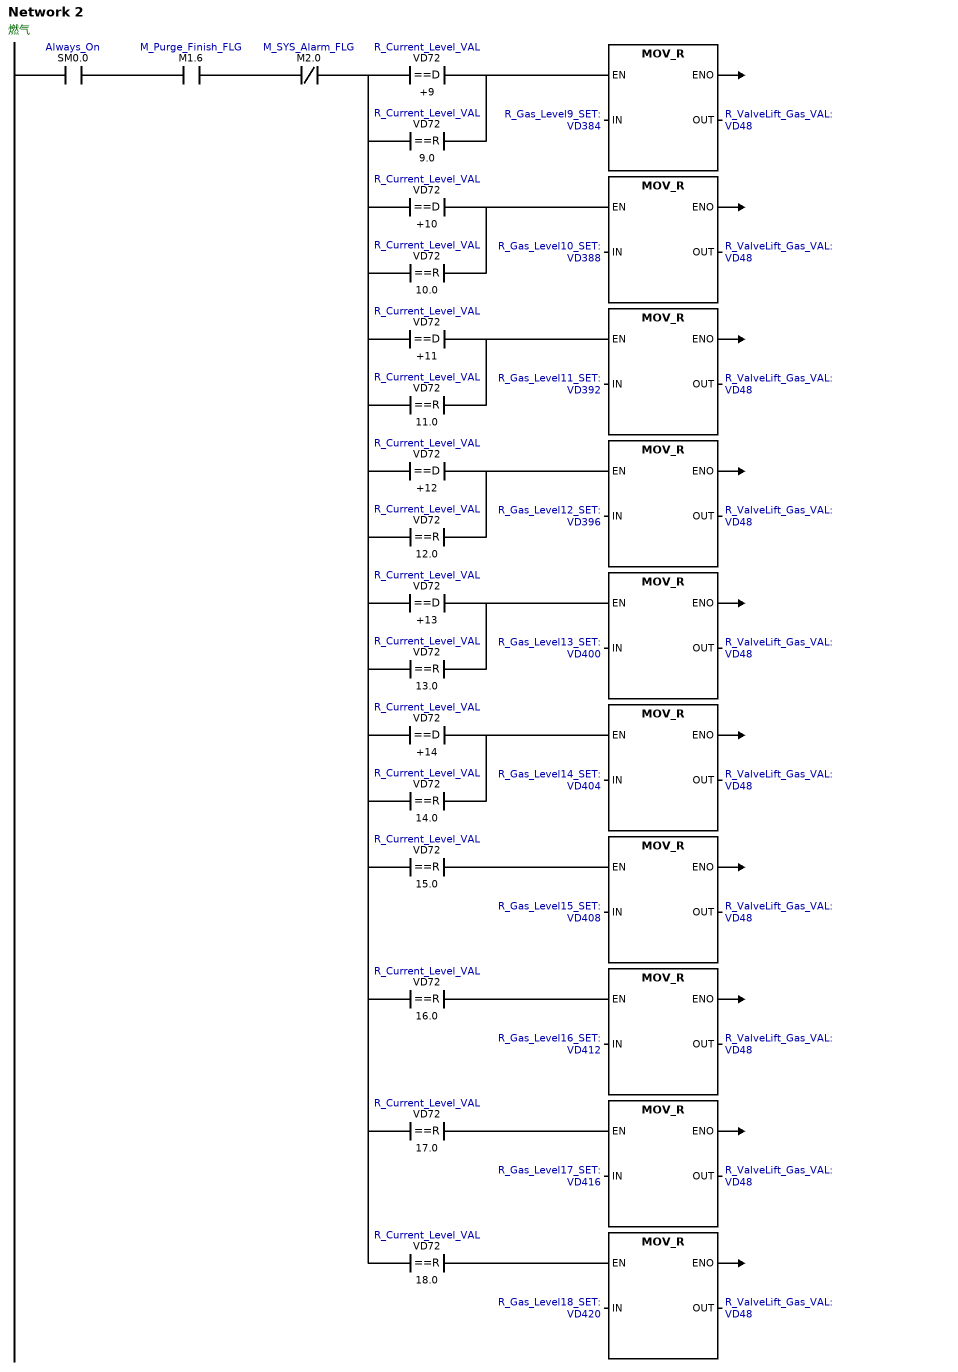
[picture p24: SBR6 networks 2-2]
Network 2
// 燃气
LD     Always_On:SM0.0
A      M_Purge_Finish_FLG:M1.6
AN     M_SYS_Alarm_FLG:M2.0
LPS
LDD=   R_Current_Level_VAL:VD72, +9
OR=    R_Current_Level_VAL:VD72, 9.0
ALD
MOVR   R_Gas_Level9_SET:VD384, R_ValveLift_Gas_VAL:VD48
LRD
LDD=   R_Current_Level_VAL:VD72, +10
OR=    R_Current_Level_VAL:VD72, 10.0
ALD
MOVR   R_Gas_Level10_SET:VD388, R_ValveLift_Gas_VAL:VD48
LRD
LDD=   R_Current_Level_VAL:VD72, +11
OR=    R_Current_Level_VAL:VD72, 11.0
ALD
MOVR   R_Gas_Level11_SET:VD392, R_ValveLift_Gas_VAL:VD48
LRD
LDD=   R_Current_Level_VAL:VD72, +12
OR=    R_Current_Level_VAL:VD72, 12.0
ALD
MOVR   R_Gas_Level12_SET:VD396, R_ValveLift_Gas_VAL:VD48
LRD
LDD=   R_Current_Level_VAL:VD72, +13
OR=    R_Current_Level_VAL:VD72, 13.0
ALD
MOVR   R_Gas_Level13_SET:VD400, R_ValveLift_Gas_VAL:VD48
LRD
LDD=   R_Current_Level_VAL:VD72, +14
OR=    R_Current_Level_VAL:VD72, 14.0
ALD
MOVR   R_Gas_Level14_SET:VD404, R_ValveLift_Gas_VAL:VD48
LPP
LPS
AR=    R_Current_Level_VAL:VD72, 15.0
MOVR   R_Gas_Level15_SET:VD408, R_ValveLift_Gas_VAL:VD48
LRD
AR=    R_Current_Level_VAL:VD72, 16.0
MOVR   R_Gas_Level16_SET:VD412, R_ValveLift_Gas_VAL:VD48
LRD
AR=    R_Current_Level_VAL:VD72, 17.0
MOVR   R_Gas_Level17_SET:VD416, R_ValveLift_Gas_VAL:VD48
LPP
AR=    R_Current_Level_VAL:VD72, 18.0
MOVR   R_Gas_Level18_SET:VD420, R_ValveLift_Gas_VAL:VD48
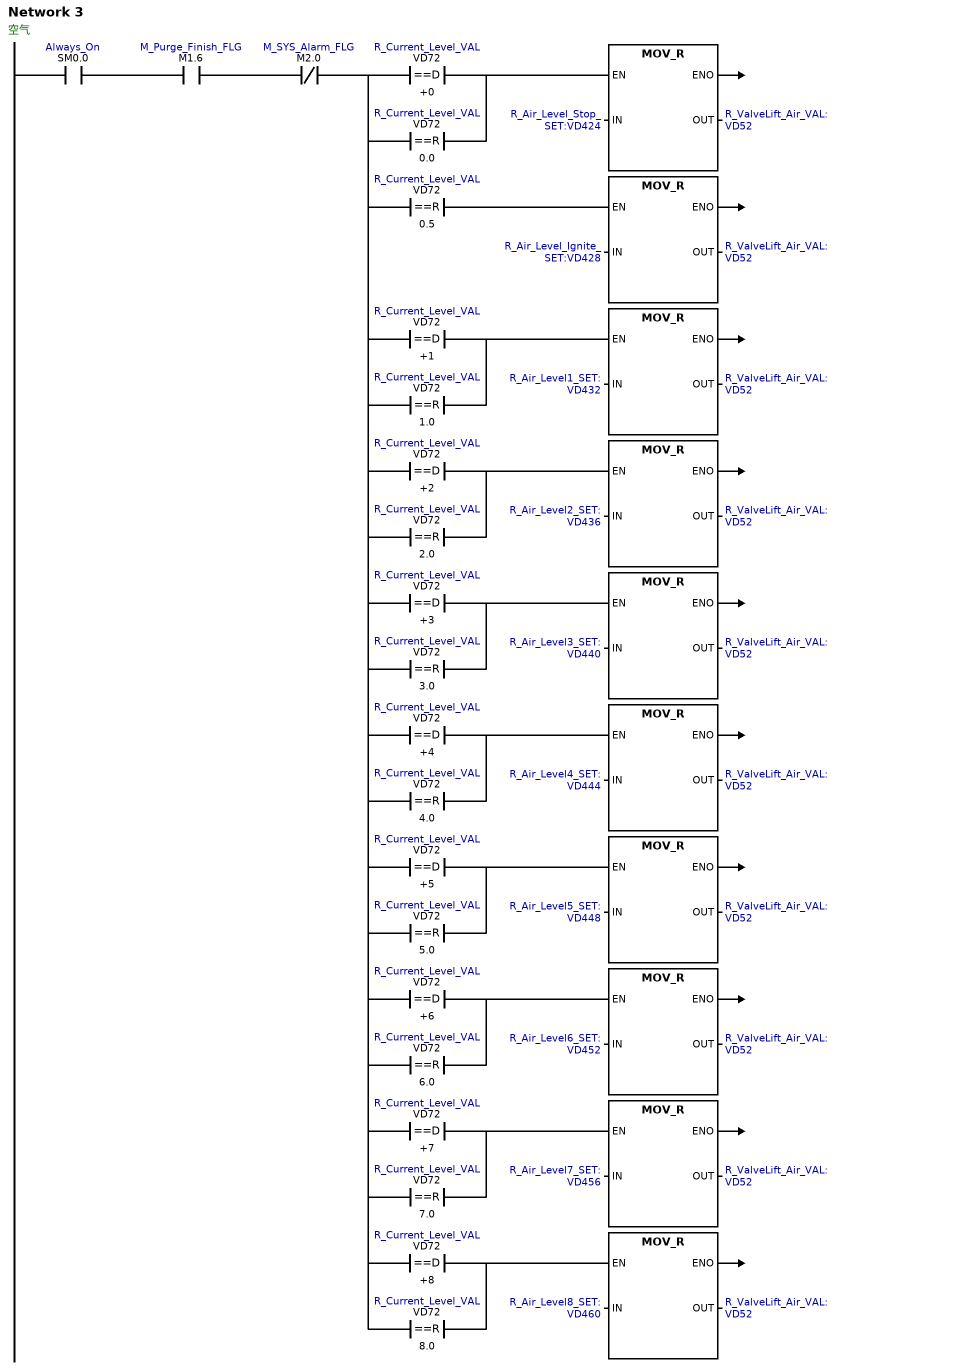
Network 3
// 空气
LD     Always_On:SM0.0
A      M_Purge_Finish_FLG:M1.6
AN     M_SYS_Alarm_FLG:M2.0
LPS
LDD=   R_Current_Level_VAL:VD72, +0
OR=    R_Current_Level_VAL:VD72, 0.0
ALD
MOVR   R_Air_Level_Stop_SET:VD424, R_ValveLift_Air_VAL:VD52
LRD
AR=    R_Current_Level_VAL:VD72, 0.5
MOVR   R_Air_Level_Ignite_SET:VD428, R_ValveLift_Air_VAL:VD52
LRD
LDD=   R_Current_Level_VAL:VD72, +1
OR=    R_Current_Level_VAL:VD72, 1.0
ALD
MOVR   R_Air_Level1_SET:VD432, R_ValveLift_Air_VAL:VD52
LRD
LDD=   R_Current_Level_VAL:VD72, +2
OR=    R_Current_Level_VAL:VD72, 2.0
ALD
MOVR   R_Air_Level2_SET:VD436, R_ValveLift_Air_VAL:VD52
LRD
LDD=   R_Current_Level_VAL:VD72, +3
OR=    R_Current_Level_VAL:VD72, 3.0
ALD
MOVR   R_Air_Level3_SET:VD440, R_ValveLift_Air_VAL:VD52
LRD
LDD=   R_Current_Level_VAL:VD72, +4
OR=    R_Current_Level_VAL:VD72, 4.0
ALD
MOVR   R_Air_Level4_SET:VD444, R_ValveLift_Air_VAL:VD52
LRD
LDD=   R_Current_Level_VAL:VD72, +5
OR=    R_Current_Level_VAL:VD72, 5.0
ALD
MOVR   R_Air_Level5_SET:VD448, R_ValveLift_Air_VAL:VD52
LRD
LDD=   R_Current_Level_VAL:VD72, +6
OR=    R_Current_Level_VAL:VD72, 6.0
ALD
MOVR   R_Air_Level6_SET:VD452, R_ValveLift_Air_VAL:VD52
LRD
LDD=   R_Current_Level_VAL:VD72, +7
OR=    R_Current_Level_VAL:VD72, 7.0
ALD
MOVR   R_Air_Level7_SET:VD456, R_ValveLift_Air_VAL:VD52
LPP
LDD=   R_Current_Level_VAL:VD72, +8
OR=    R_Current_Level_VAL:VD72, 8.0
ALD
MOVR   R_Air_Level8_SET:VD460, R_ValveLift_Air_VAL:VD52
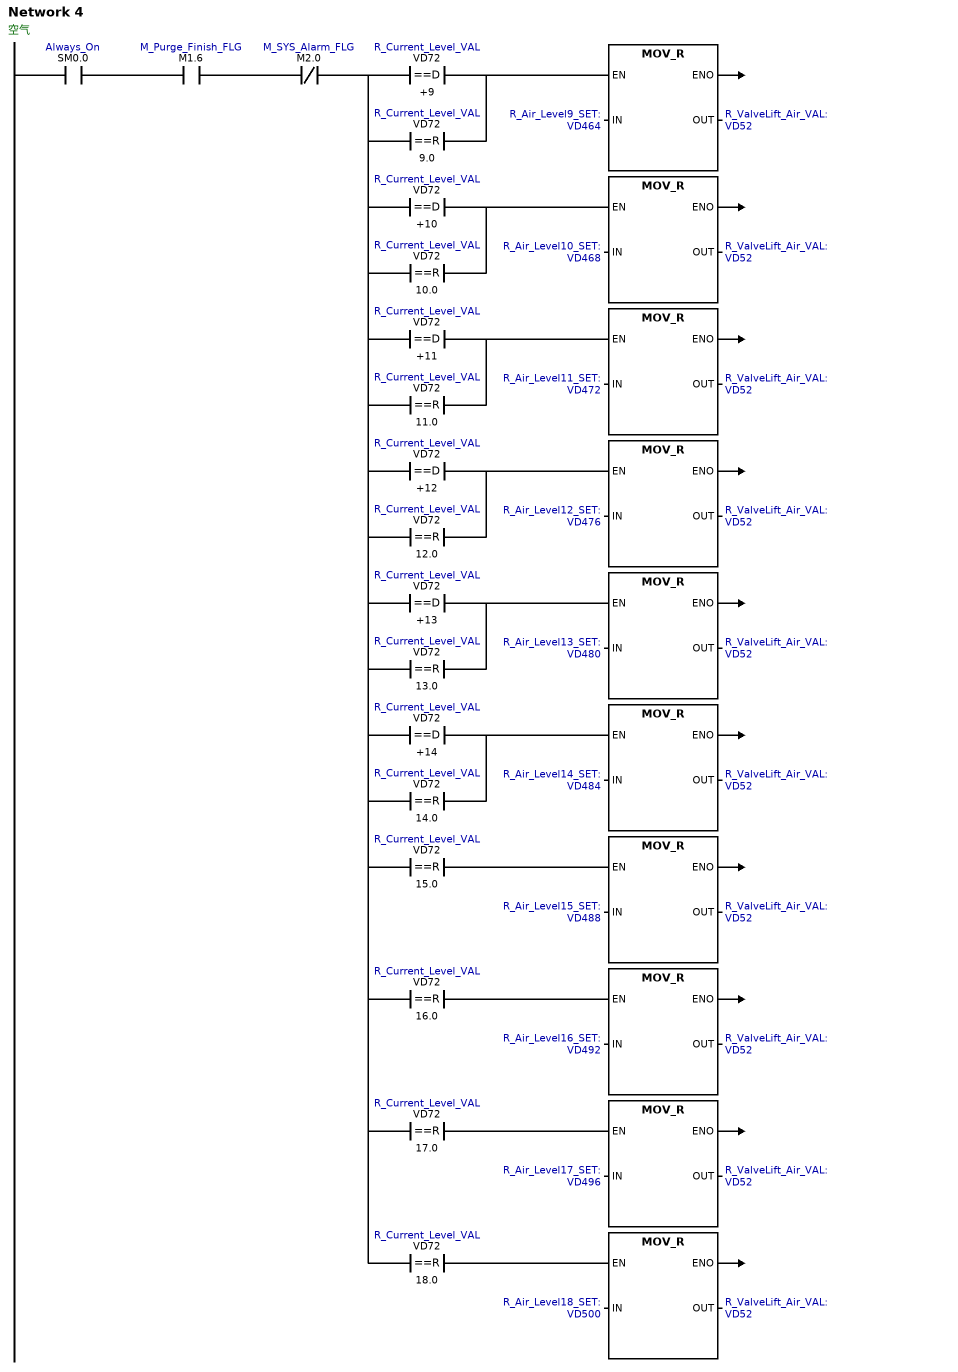
Network 4
// 空气
LD     Always_On:SM0.0
A      M_Purge_Finish_FLG:M1.6
AN     M_SYS_Alarm_FLG:M2.0
LPS
LDD=   R_Current_Level_VAL:VD72, +9
OR=    R_Current_Level_VAL:VD72, 9.0
ALD
MOVR   R_Air_Level9_SET:VD464, R_ValveLift_Air_VAL:VD52
LRD
LDD=   R_Current_Level_VAL:VD72, +10
OR=    R_Current_Level_VAL:VD72, 10.0
ALD
MOVR   R_Air_Level10_SET:VD468, R_ValveLift_Air_VAL:VD52
LRD
LDD=   R_Current_Level_VAL:VD72, +11
OR=    R_Current_Level_VAL:VD72, 11.0
ALD
MOVR   R_Air_Level11_SET:VD472, R_ValveLift_Air_VAL:VD52
LRD
LDD=   R_Current_Level_VAL:VD72, +12
OR=    R_Current_Level_VAL:VD72, 12.0
ALD
MOVR   R_Air_Level12_SET:VD476, R_ValveLift_Air_VAL:VD52
LRD
LDD=   R_Current_Level_VAL:VD72, +13
OR=    R_Current_Level_VAL:VD72, 13.0
ALD
MOVR   R_Air_Level13_SET:VD480, R_ValveLift_Air_VAL:VD52
LRD
LDD=   R_Current_Level_VAL:VD72, +14
OR=    R_Current_Level_VAL:VD72, 14.0
ALD
MOVR   R_Air_Level14_SET:VD484, R_ValveLift_Air_VAL:VD52
LPP
LPS
AR=    R_Current_Level_VAL:VD72, 15.0
MOVR   R_Air_Level15_SET:VD488, R_ValveLift_Air_VAL:VD52
LRD
AR=    R_Current_Level_VAL:VD72, 16.0
MOVR   R_Air_Level16_SET:VD492, R_ValveLift_Air_VAL:VD52
LRD
AR=    R_Current_Level_VAL:VD72, 17.0
MOVR   R_Air_Level17_SET:VD496, R_ValveLift_Air_VAL:VD52
LPP
AR=    R_Current_Level_VAL:VD72, 18.0
MOVR   R_Air_Level18_SET:VD500, R_ValveLift_Air_VAL:VD52
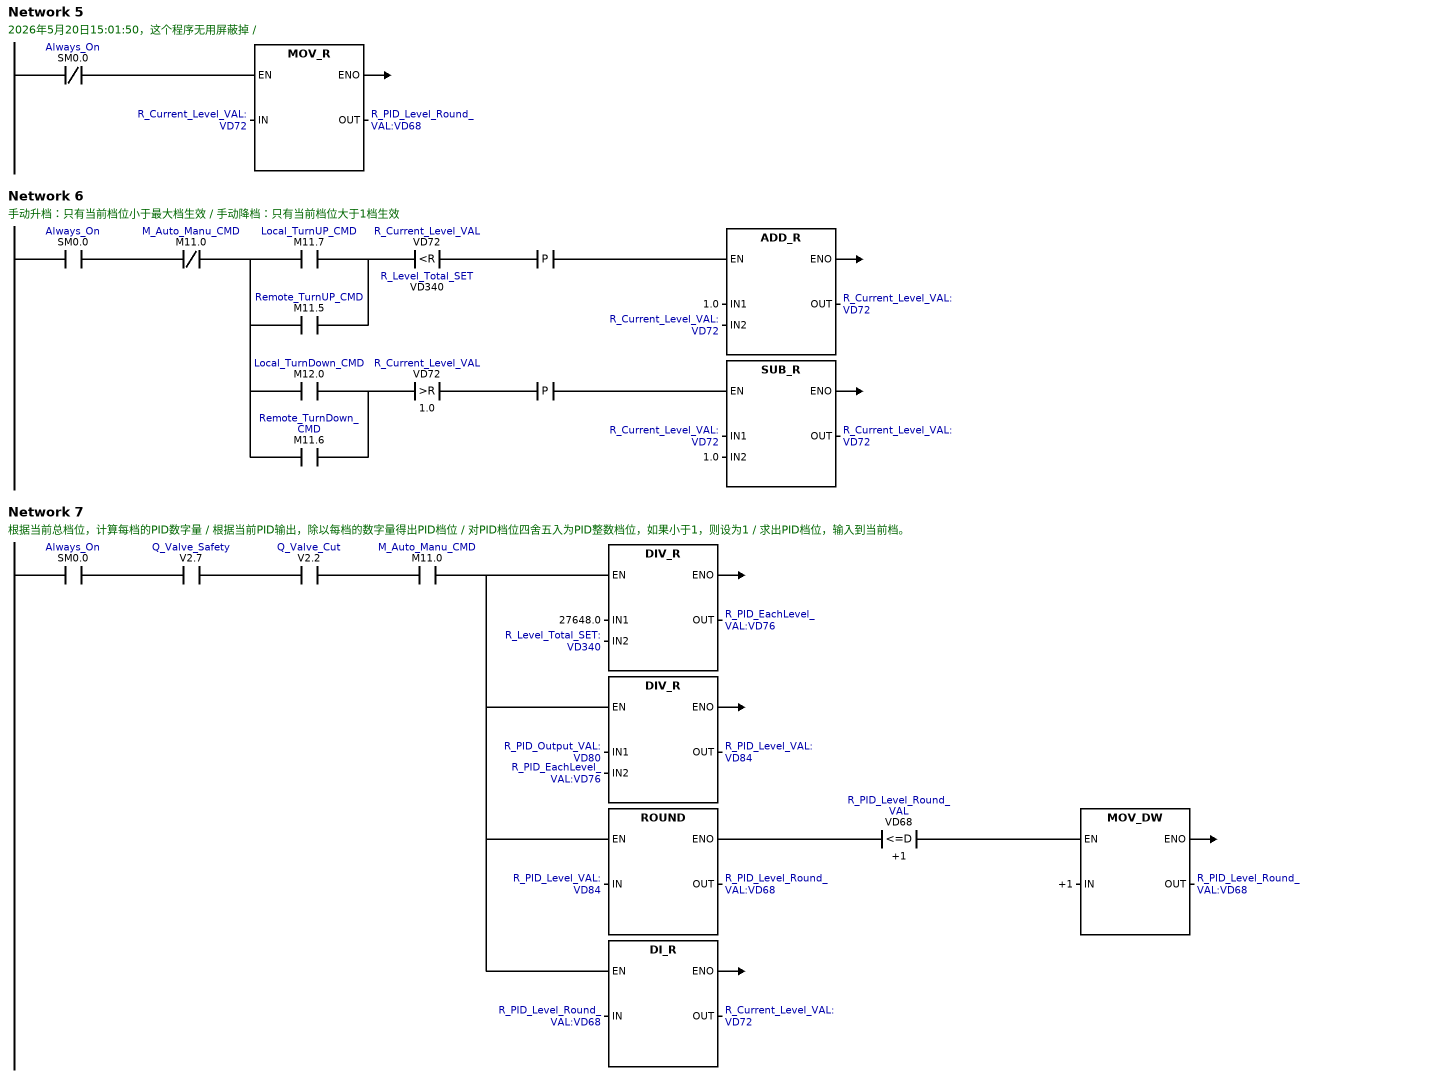
Network 5
// 2026年5月20日15:01:50，这个程序无用屏蔽掉
// 
LDN    Always_On:SM0.0
MOVR   R_Current_Level_VAL:VD72, R_PID_Level_Round_VAL:VD68
Network 6
// 手动升档：只有当前档位小于最大档生效
// 手动降档：只有当前档位大于1档生效
LD     Always_On:SM0.0
AN     M_Auto_Manu_CMD:M11.0
LPS
LD     Local_TurnUP_CMD:M11.7
O      Remote_TurnUP_CMD:M11.5
ALD
AR<    R_Current_Level_VAL:VD72, R_Level_Total_SET:VD340
EU
+R     1.0, R_Current_Level_VAL:VD72
LPP
LD     Local_TurnDown_CMD:M12.0
O      Remote_TurnDown_CMD:M11.6
ALD
AR>    R_Current_Level_VAL:VD72, 1.0
EU
-R     1.0, R_Current_Level_VAL:VD72
Network 7
// 根据当前总档位，计算每档的PID数字量
// 根据当前PID输出，除以每档的数字量得出PID档位
// 对PID档位四舍五入为PID整数档位，如果小于1，则设为1
// 求出PID档位，输入到当前档。
LD     Always_On:SM0.0
A      Q_Valve_Safety:V2.7
A      Q_Valve_Cut:V2.2
A      M_Auto_Manu_CMD:M11.0
LPS
MOVR   27648.0, R_PID_EachLevel_VAL:VD76
/R     R_Level_Total_SET:VD340, R_PID_EachLevel_VAL:VD76
MOVR   R_PID_Output_VAL:VD80, R_PID_Level_VAL:VD84
/R     R_PID_EachLevel_VAL:VD76, R_PID_Level_VAL:VD84
ROUND  R_PID_Level_VAL:VD84, R_PID_Level_Round_VAL:VD68
AENO
AD<=   R_PID_Level_Round_VAL:VD68, +1
MOVD   +1, R_PID_Level_Round_VAL:VD68
LPP
DTR    R_PID_Level_Round_VAL:VD68, R_Current_Level_VAL:VD72
END_SUBROUTINE_BLOCK

SUBROUTINE_BLOCK 远程通讯:SBR7
TITLE=远程通讯子程序
// 功能：
// 1、初始化从站（PLC）
// 	模式Mode（通讯协议）：	1、Modubs协议；0、PPI协
// 	地址Addr	：	1-247
// 	波特率Baud：	1200、2400、4800、9600、19200、38400、57600、11500
// 	奇偶校验Parity：	0无校验、1奇校验、2偶校验
// 	端口Port：	0=CPU集成RS-485端口，1=可选信号板上的RS-485或RS-232
// 	延时Delay：	可以是0-32767
// 	MaxIQ：		设置Modbus地址0XXXX和1XXXX可用 的I和Q点数，0-256
// 	MaxAI：		设置Modbus地址3XXXX可用的字输入（AI）寄存器数，0（CR系列）或56（其它系列）
// 	MaxHold：	设置Modbus地址4XXXX或4yyyyy可访问的V存储器中的字保持寄存器数。如果要允许 Modbus 主站访问 2000 个字节的 V 存储器，请将 MaxHold的值设置为 1000 个字（保持寄存器）
// 	HoldStart：	是 V 存储器中保持寄存器的起始地址	
// 
// 2、处理主站请求
// 在每次扫描处理主站请求
// 
// 
// 
// 3、显示设备状态：
// 	故障状态RTU
// 	自动状态RTU
// 	启动状态RTU
// 	停止状态RTU
// 	本地远程状态RTU
// 
// 4、处理DCS传送过来的温度数据,VW1898
BEGIN
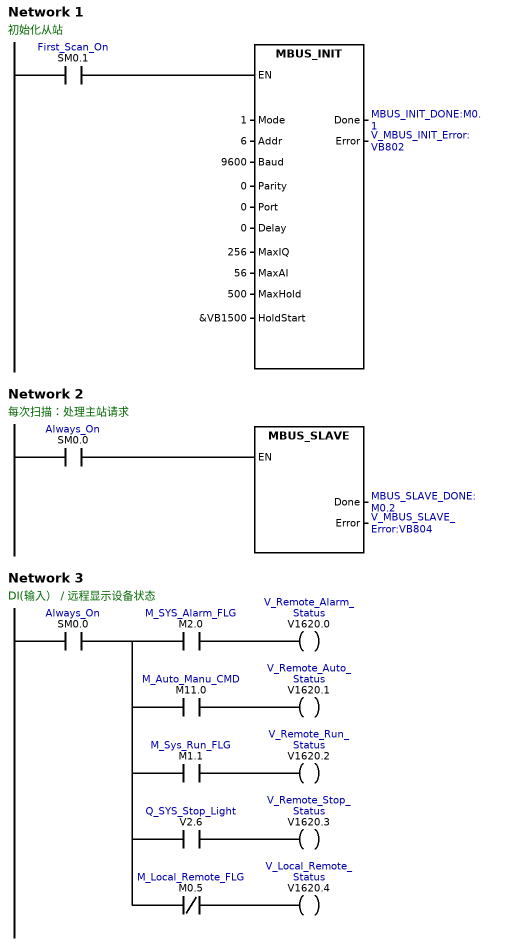
Network 1
// 初始化从站
LD     First_Scan_On:SM0.1
CALL   MBUS_INIT:SBR21, 1, 6, 9600, 0, 0, 0, 256, 56, 500, &VB1500, MBUS_INIT_DONE:M0.1, V_MBUS_INIT_Error:VB802
Network 2
// 每次扫描：处理主站请求
LD     Always_On:SM0.0
CALL   MBUS_SLAVE:SBR22, MBUS_SLAVE_DONE:M0.2, V_MBUS_SLAVE_Error:VB804
Network 3
// DI(输入）
// 远程显示设备状态
LD     Always_On:SM0.0
LPS
A      M_SYS_Alarm_FLG:M2.0
=      V_Remote_Alarm_Status:V1620.0
LRD
A      M_Auto_Manu_CMD:M11.0
=      V_Remote_Auto_Status:V1620.1
LRD
A      M_Sys_Run_FLG:M1.1
=      V_Remote_Run_Status:V1620.2
LRD
A      Q_SYS_Stop_Light:V2.6
=      V_Remote_Stop_Status:V1620.3
LPP
AN     M_Local_Remote_FLG:M0.5
=      V_Local_Remote_Status:V1620.4
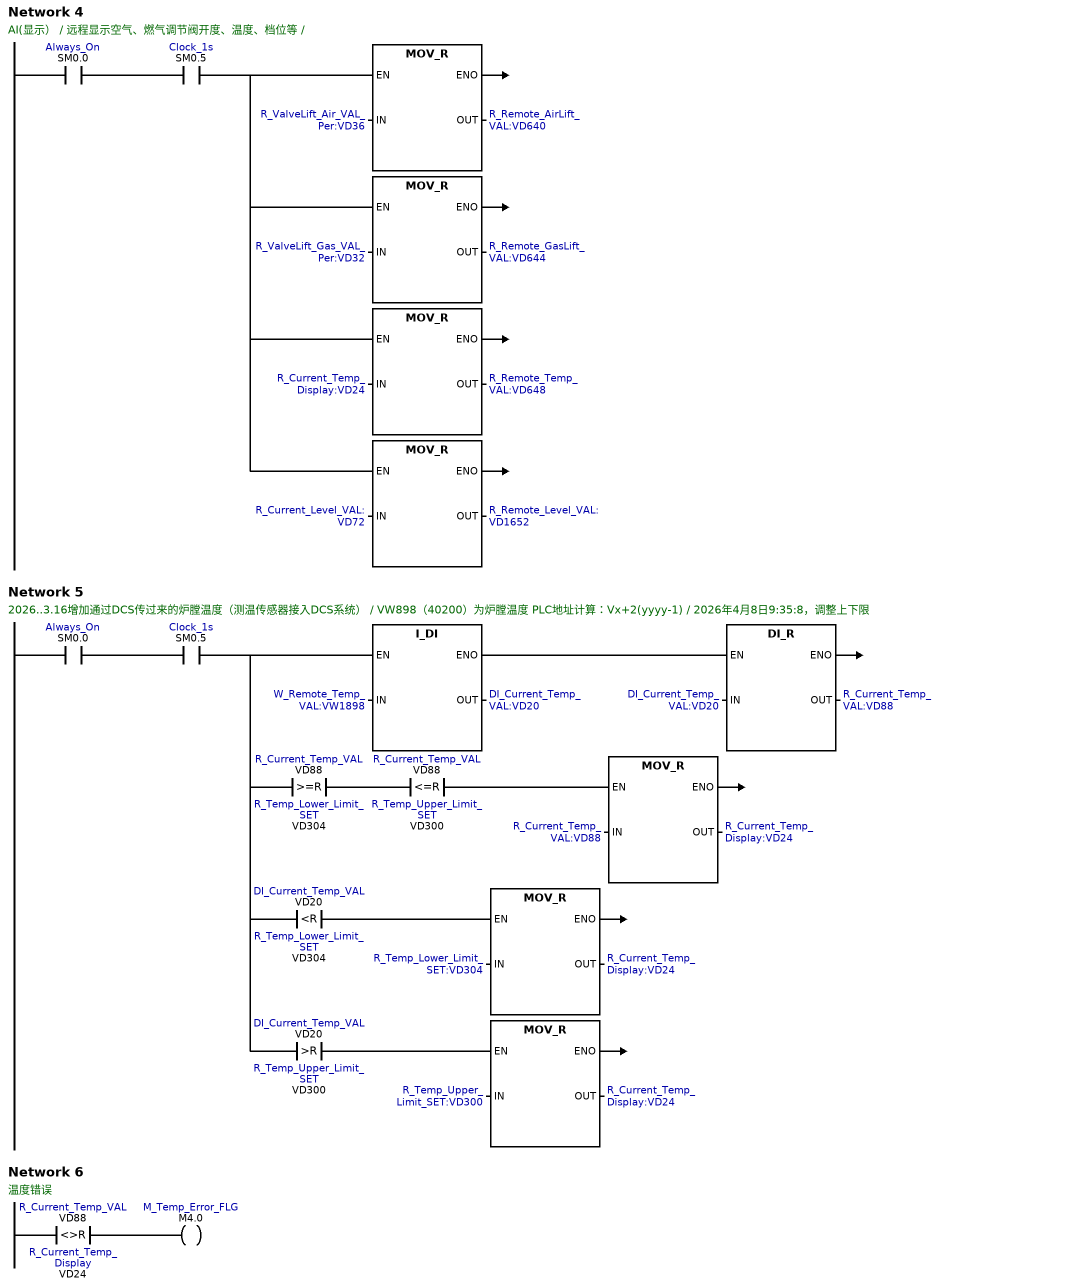
Network 4
// AI(显示）
// 远程显示空气、燃气调节阀开度、温度、档位等
// 
LD     Always_On:SM0.0
A      Clock_1s:SM0.5
MOVR   R_ValveLift_Air_VAL_Per:VD36, R_Remote_AirLift_VAL:VD640
MOVR   R_ValveLift_Gas_VAL_Per:VD32, R_Remote_GasLift_VAL:VD644
MOVR   R_Current_Temp_Display:VD24, R_Remote_Temp_VAL:VD648
MOVR   R_Current_Level_VAL:VD72, R_Remote_Level_VAL:VD1652
Network 5
// 2026..3.16增加通过DCS传过来的炉膛温度（测温传感器接入DCS系统）
// VW898（40200）为炉膛温度 PLC地址计算：Vx+2(yyyy-1)
// 2026年4月8日9:35:8，调整上下限
LD     Always_On:SM0.0
A      Clock_1s:SM0.5
LPS
ITD    W_Remote_Temp_VAL:VW1898, DI_Current_Temp_VAL:VD20
AENO
DTR    DI_Current_Temp_VAL:VD20, R_Current_Temp_VAL:VD88
LRD
AR>=   R_Current_Temp_VAL:VD88, R_Temp_Lower_Limit_SET:VD304
AR<=   R_Current_Temp_VAL:VD88, R_Temp_Upper_Limit_SET:VD300
MOVR   R_Current_Temp_VAL:VD88, R_Current_Temp_Display:VD24
LRD
AR<    DI_Current_Temp_VAL:VD20, R_Temp_Lower_Limit_SET:VD304
MOVR   R_Temp_Lower_Limit_SET:VD304, R_Current_Temp_Display:VD24
LPP
AR>    DI_Current_Temp_VAL:VD20, R_Temp_Upper_Limit_SET:VD300
MOVR   R_Temp_Upper_Limit_SET:VD300, R_Current_Temp_Display:VD24
Network 6
// 温度错误
LDR<>  R_Current_Temp_VAL:VD88, R_Current_Temp_Display:VD24
=      M_Temp_Error_FLG:M4.0
END_SUBROUTINE_BLOCK

SUBROUTINE_BLOCK IO设备:SBR8
TITLE=子程序注释
// 1、IO映射
// 2、统一输出
// 	蜂鸣器
// 	点火阀
// 	主火阀V2
// 	点火变压器
// 	有火指示灯
// 	启动指示灯
// 	停止指示灯
// 	安全阀V1
// 
// 
BEGIN
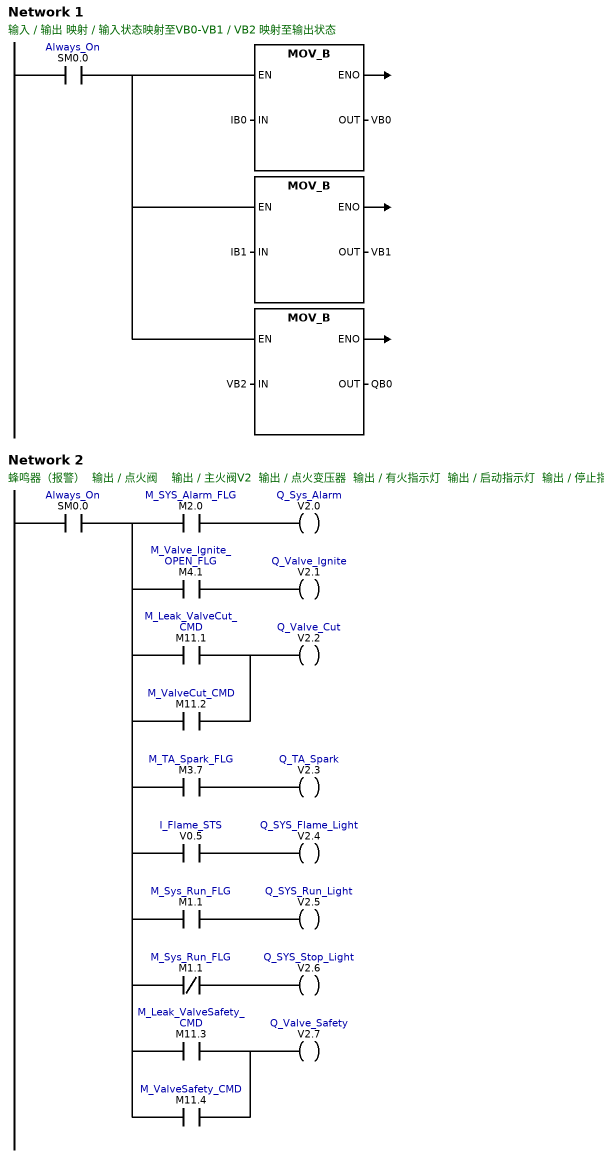
Network 1
// 输入 / 输出 映射
// 输入状态映射至VB0-VB1
// VB2 映射至输出状态
LD     Always_On:SM0.0
MOVB   IB0, VB0
MOVB   IB1, VB1
MOVB   VB2, QB0
Network 2
// 蜂鸣器（报警）	输出
// 点火阀		输出
// 主火阀V2	输出
// 点火变压器	输出
// 有火指示灯	输出
// 启动指示灯	输出
// 停止指示灯	输出
// 安全阀V1	输出
// 
LD     Always_On:SM0.0
LPS
A      M_SYS_Alarm_FLG:M2.0
=      Q_Sys_Alarm:V2.0
LRD
A      M_Valve_Ignite_OPEN_FLG:M4.1
=      Q_Valve_Ignite:V2.1
LRD
LD     M_Leak_ValveCut_CMD:M11.1
O      M_ValveCut_CMD:M11.2
ALD
=      Q_Valve_Cut:V2.2
LRD
LPS
A      M_TA_Spark_FLG:M3.7
=      Q_TA_Spark:V2.3
LRD
A      I_Flame_STS:V0.5
=      Q_SYS_Flame_Light:V2.4
LRD
A      M_Sys_Run_FLG:M1.1
=      Q_SYS_Run_Light:V2.5
LPP
AN     M_Sys_Run_FLG:M1.1
=      Q_SYS_Stop_Light:V2.6
LPP
LD     M_Leak_ValveSafety_CMD:M11.3
O      M_ValveSafety_CMD:M11.4
ALD
=      Q_Valve_Safety:V2.7
END_SUBROUTINE_BLOCK

SUBROUTINE_BLOCK 运行时间:SBR9
TITLE=
BEGIN
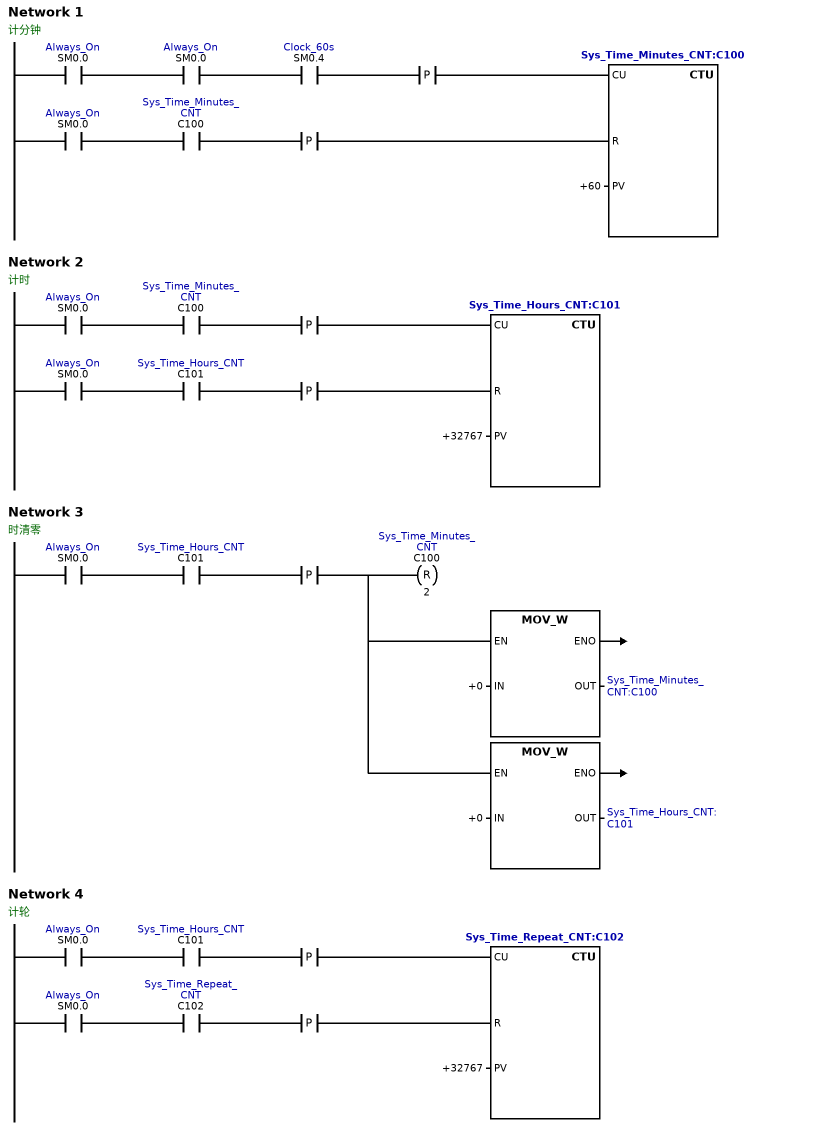
Network 1
// 计分钟
LD     Always_On:SM0.0
A      Always_On:SM0.0
A      Clock_60s:SM0.4
EU
LD     Always_On:SM0.0
A      Sys_Time_Minutes_CNT:C100
EU
CTU    Sys_Time_Minutes_CNT:C100, +60
Network 2
// 计时
LD     Always_On:SM0.0
A      Sys_Time_Minutes_CNT:C100
EU
LD     Always_On:SM0.0
A      Sys_Time_Hours_CNT:C101
EU
CTU    Sys_Time_Hours_CNT:C101, +32767
Network 3
// 时清零
LD     Always_On:SM0.0
A      Sys_Time_Hours_CNT:C101
EU
R      Sys_Time_Minutes_CNT:C100, 2
MOVW   +0, Sys_Time_Minutes_CNT:C100
MOVW   +0, Sys_Time_Hours_CNT:C101
Network 4
// 计轮
LD     Always_On:SM0.0
A      Sys_Time_Hours_CNT:C101
EU
LD     Always_On:SM0.0
A      Sys_Time_Repeat_CNT:C102
EU
CTU    Sys_Time_Repeat_CNT:C102, +32767
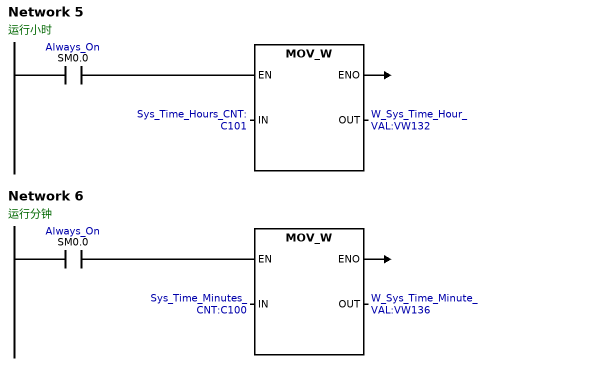
Network 5
// 运行小时
LD     Always_On:SM0.0
MOVW   Sys_Time_Hours_CNT:C101, W_Sys_Time_Hour_VAL:VW132
Network 6
// 运行分钟
LD     Always_On:SM0.0
MOVW   Sys_Time_Minutes_CNT:C100, W_Sys_Time_Minute_VAL:VW136
END_SUBROUTINE_BLOCK

SUBROUTINE_BLOCK 报警复位:SBR13
TITLE=报警复位子程序
// 功能：
// 1、报警逻辑
// 系统故障报警停机如：	
// 	检漏报警		停机
// 	空气压力低报警		停机
// 	燃气压力高报警		停机
// 	燃气压力低报警		停机
// 	点火前检测到火焰报警	停机
// 	点火失败报警		停机
// 	火焰丢失报警		停机
// 关闭所有燃气阀门：包括点火阀、主火阀、安全阀、
// 复位点火成功标志，
// 
// 调节阀故障只显示
// 	空气调节阀检测失败报警	提示
// 	燃气调节阀检测失败报警	提示
// 
// 
// 2、复位逻辑
// 复位7个故障，M20.1-M20.7
// 
// 两个调节阀故障，上电的时候才复位，这里不复位。
// 
// 
// 
BEGIN
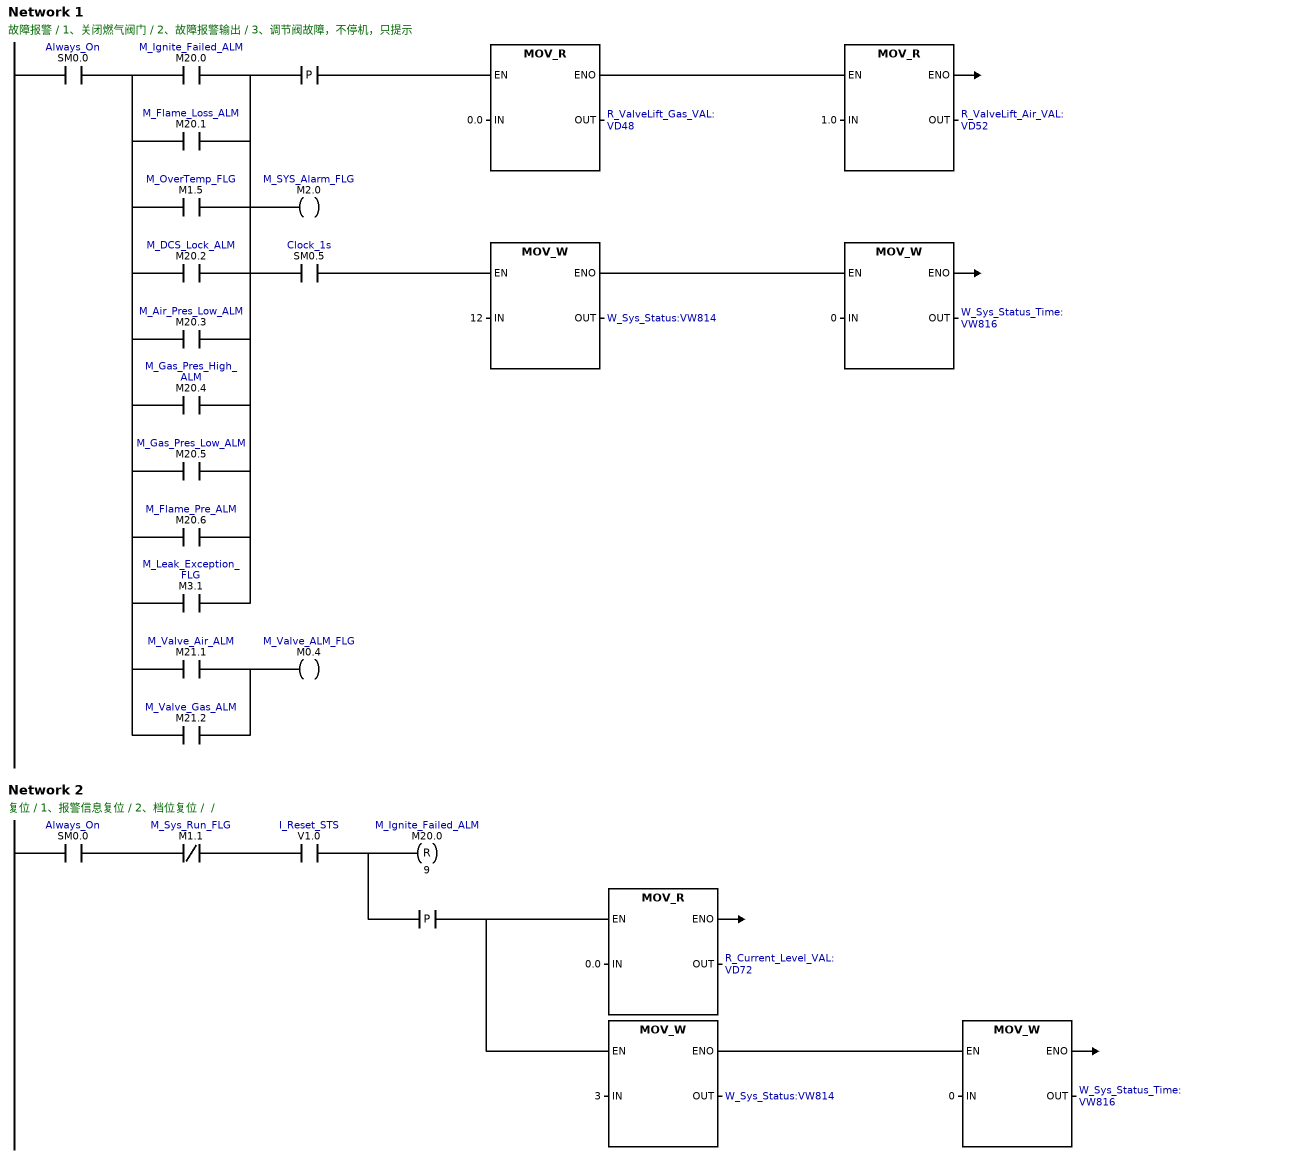
Network 1
// 故障报警
// 1、关闭燃气阀门
// 2、故障报警输出
// 3、调节阀故障，不停机，只提示
LD     Always_On:SM0.0
LPS
LD     M_Ignite_Failed_ALM:M20.0
O      M_Flame_Loss_ALM:M20.1
O      M_OverTemp_FLG:M1.5
O      M_DCS_Lock_ALM:M20.2
O      M_Air_Pres_Low_ALM:M20.3
O      M_Gas_Pres_High_ALM:M20.4
O      M_Gas_Pres_Low_ALM:M20.5
O      M_Flame_Pre_ALM:M20.6
O      M_Leak_Exception_FLG:M3.1
ALD
LPS
EU
MOVR   0.0, R_ValveLift_Gas_VAL:VD48
AENO
MOVR   1.0, R_ValveLift_Air_VAL:VD52
LRD
=      M_SYS_Alarm_FLG:M2.0
LPP
A      Clock_1s:SM0.5
MOVW   12, W_Sys_Status:VW814
AENO
MOVW   0, W_Sys_Status_Time:VW816
LPP
LD     M_Valve_Air_ALM:M21.1
O      M_Valve_Gas_ALM:M21.2
ALD
=      M_Valve_ALM_FLG:M0.4
Network 2
// 复位
// 1、报警信息复位
// 2、档位复位
// 
// 
LD     Always_On:SM0.0
AN     M_Sys_Run_FLG:M1.1
A      I_Reset_STS:V1.0
R      M_Ignite_Failed_ALM:M20.0, 9
EU
MOVR   0.0, R_Current_Level_VAL:VD72
MOVW   3, W_Sys_Status:VW814
AENO
MOVW   0, W_Sys_Status_Time:VW816
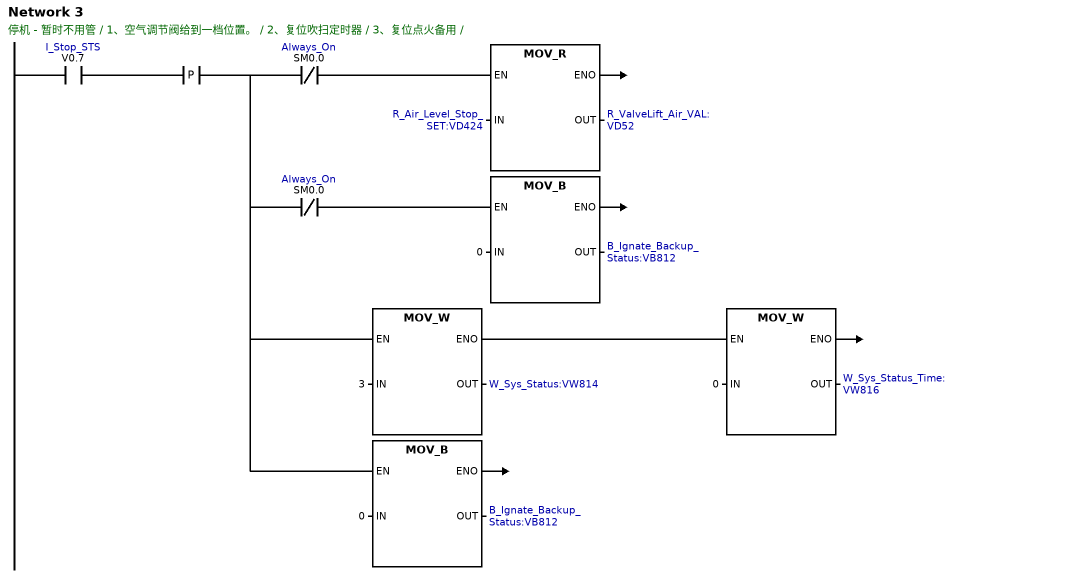
Network 3
// 停机 - 暂时不用管
// 1、空气调节阀给到一档位置。
// 2、复位吹扫定时器
// 3、复位点火备用
// 
LD     I_Stop_STS:V0.7
EU
LPS
AN     Always_On:SM0.0
MOVR   R_Air_Level_Stop_SET:VD424, R_ValveLift_Air_VAL:VD52
LRD
AN     Always_On:SM0.0
MOVB   0, B_Ignate_Backup_Status:VB812
LRD
MOVW   3, W_Sys_Status:VW814
AENO
MOVW   0, W_Sys_Status_Time:VW816
LPP
MOVB   0, B_Ignate_Backup_Status:VB812
END_SUBROUTINE_BLOCK

// SBR18: protected block, not included

// SBR21: protected block, not included

// SBR22: protected block, not included

// SBR23: protected block, not included

// SBR24: protected block, not included

// SBR30: protected block, not included

// SBR31: protected block, not included

// INT0: protected block, not included

DATA_BLOCK_TAB 页面_1
BEGIN
//数据页注释
//按 F1 获取帮助和示例数据页
         R_Stage1_Temp_SET, 0.0
         R_Stage2_Temp_SET, 0.0
         R_Stage3_Temp_SET, 0.0
         R_Stage4_Temp_SET, 0.0
         R_Stage5_Temp_SET, 0.0
         R_Stage6_Temp_SET, 500.0
         W_Stage1_Temp_Time_SET, 0
         W_Stage2_Temp_Time_SET, 0
         W_Stage3_Temp_Time_SET, 0
         W_Stage4_Temp_Time_SET, 0
         W_Stage5_Temp_Time_SET, 0
         W_Stage6_Temp_Time_SET, 1
         R_Temp_Upper_Limit_SET, 999.0
         R_Over_Temp_Stop_SET, 985.0
         R_PID_P_SET, 17.0
         R_PID_I_SET, 10.0
         R_PID_D_SET, 0
         R_PID_Ts_SET, 0.01
         R_Gas_Level1_SET, 15.0
         R_Gas_Level2_SET, 20.0
         R_Gas_Level3_SET, 25.0
         R_Gas_Level4_SET, 30.0
         R_Gas_Level5_SET, 35.0
         R_Gas_Level6_SET, 40.0
         R_Gas_Level7_SET, 45.0
         R_Gas_Level8_SET, 50.0
         R_Gas_Level9_SET, 55.0
         R_Gas_Level10_SET, 60.0
         R_Gas_Level11_SET, 65.0
         R_Gas_Level12_SET, 70.0
         R_Gas_Level13_SET, 75.0
         R_Gas_Level14_SET, 80.0
         R_Air_Level1_SET, 15.0
         R_Air_Level2_SET, 20.0
         R_Air_Level3_SET, 25.0
         R_Air_Level4_SET, 30.0
         R_Air_Level5_SET, 35.0
         R_Air_Level6_SET, 40.0
         R_Air_Level7_SET, 45.0
         R_Air_Level8_SET, 50.0
         R_Air_Level9_SET, 55.0
         R_Air_Level10_SET, 60.0
         R_Air_Level11_SET, 65.0
         R_Air_Level12_SET, 70.0
         R_Air_Level13_SET, 75.0
         R_Air_Level14_SET, 80.0
         R_Level_Total_SET, 14.0
VD564    80.0
         R_Air_Level_Ignite_SET, 10.0
         W_Ignite_Delay_SET, 9
         W_ValveCut_Delay_SET, 9
END_DATA_BLOCK_TAB
